// TIA Portal V16 export
// export: Created 2022-11-17T15:49:36.4302369Z, ExportSetting WithDefaults, DisplayName Totally Integrated Automation Portal, DisplayVersion V16 Update 6, DisplayName TIA Portal Version Control Interface, DisplayVersion V16 Update 2, DisplayName TIA Portal Openness, DisplayVersion V16 Update 6, DisplayName SINAMICS Startdrive Advanced, DisplayVersion V16 Update 5, DisplayName SINAMICS Startdrive G130, G150, S120, S150, SINAMICS MV, S210, DisplayVersion V16 Update 5, DisplayName SINAMICS Startdrive G110M, G120, G120C, G120D, G120P, G115D, DisplayVersion V16 Update 5, DisplayName STEP 7 Professional, DisplayVersion V16 Update 6, DisplayName STEP 7 Safety, DisplayVersion V16, DisplayName WinCC Advanced, DisplayVersion V16 Update 6
DATA_BLOCK "DB04_Conveyor"   // DB4
{ S7_Optimized_Access := 'FALSE' }
AUTHOR : Robopac
VERSION : 0.0
// stored: AutoNumber false, IsOnlyStoredInLoadMemory false, IsWriteProtectedInAS false
   VAR RETAIN
      dbw0 : Int := 0;
      dbw2 : Int := 0;
      dbx4_0 : Bool := TRUE;   // Pallet positioned
      dbx4_1 : Bool := FALSE;   // Deceleration for pallet positioning
      dbx4_2 : Bool := FALSE;   // Support memory for wrong pallet positioning emergency
      dbx4_3 : Bool := FALSE;   // Unload memory for outfeed conveyor
      dbx4_4 : Bool := TRUE;   // Support for end of transfer signal for pallet load/unload
      dbx4_5 : Bool := TRUE;   // Short pallet positioned
      dbx4_6 : Bool := TRUE;   // Pallet positioned for clampcutcycle
      dbx4_7 : Bool := FALSE;   // Pallet positioned from reverse
      dbb5 : Byte := 16#00;
      dbw6 : Int := 0;
      dbw8 : Int := 0;
      dbw10 : Int := 0;   // Pallet lenght measured in infeed (pulse)
      dbw12 : Int := 0;   // Pallet lenght measured in central machine (pulse)
      dbw14 : Int := 0;   // Pallet lenght measured in infeed (mm)
      dbw16 : Int := 0;   // Pallet lenght measured in central machine (mm)
      dbw18 : Int := 0;   // Half pallet lenght for selfcentering system
      dbw20 : Int := -100;   // Deceleration for pallet positioning on selfcentering system
      dbw22 : Int := 78;   // Support for conveyor movement speed
      dbw24 : Int := 0;
      dbw26 : Int := 0;
      dbw28 : Int := 0;
      dbw30 : Int := 0;
      dbw32 : Int := 0;
      dbw34 : Int := 0;
      dbd36 : DInt := 0;
      dbd40 : DInt := 0;
      dbd44 : DInt := 0;
      dbd48 : DInt := 0;
      dbd52 : DInt := 0;
      dbd56 : DInt := 0;
      dbd60 : DInt := 0;
      dbd64 : DInt := 0;
      dbd68 : DInt := 0;
      dbd72 : DInt := 0;
      dbw76 : Int := 0;
      dbb78 : Byte := 16#00;   // Rope unit for running spool carriage height (1=Excluded 2=Inc 3=Inc during
      dbb79 : Byte := 16#00;   // Rope unit for running spool carriage height (1=Excluded 2=Inc 3=Inc during
      dbd80 : DInt := 0;
      dbd84 : DInt := 0;
   END_VAR
BEGIN
END_DATA_BLOCK
